// Mitsubishi GX Works2 project: atuo   PLC: FX3U/FX3UC

PROGRAM MAIN
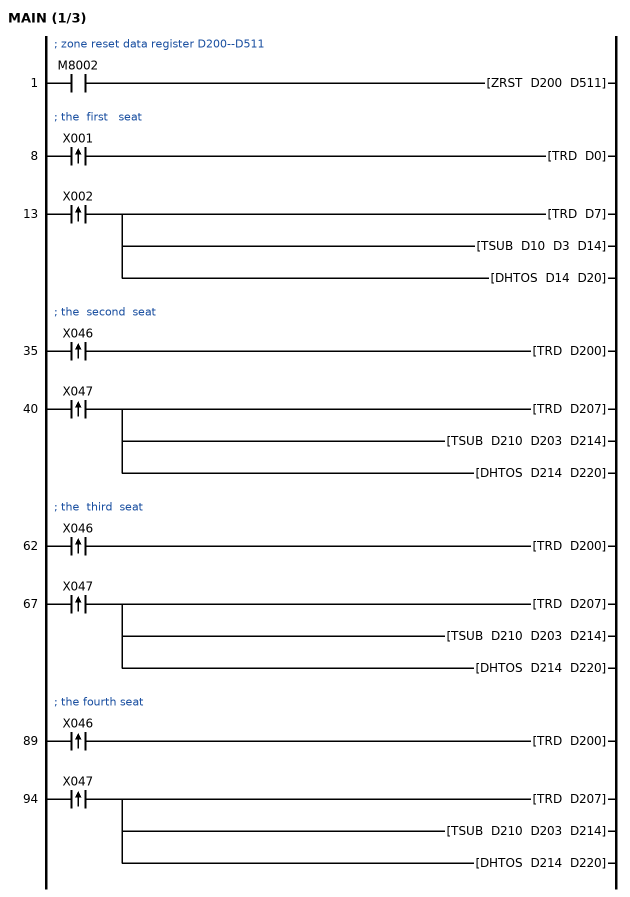
; zone reset data register D200--D511
1     LD      M8002
      ZRST    D200 D511
; the  first   seat
8     LDP     X001
      TRD     D0
13    LDP     X002
      TRD     D7
      TSUB    D10 D3 D14
      DHTOS   D14 D20
; the  second  seat
35    LDP     X046
      TRD     D200
40    LDP     X047
      TRD     D207
      TSUB    D210 D203 D214
      DHTOS   D214 D220
; the  third  seat
62    LDP     X046
      TRD     D200
67    LDP     X047
      TRD     D207
      TSUB    D210 D203 D214
      DHTOS   D214 D220
; the fourth seat
89    LDP     X046
      TRD     D200
94    LDP     X047
      TRD     D207
      TSUB    D210 D203 D214
      DHTOS   D214 D220
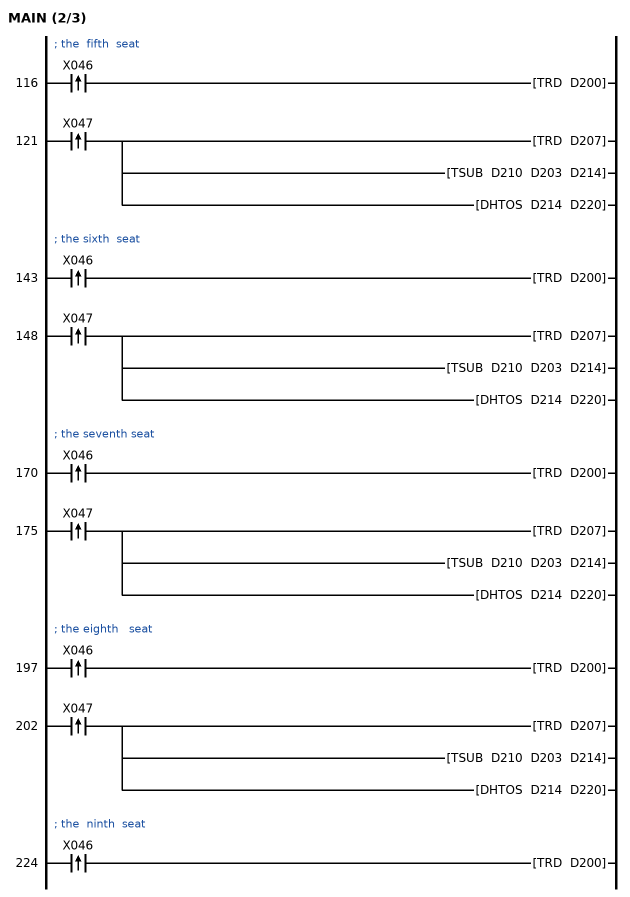
; the  fifth  seat
116   LDP     X046
      TRD     D200
121   LDP     X047
      TRD     D207
      TSUB    D210 D203 D214
      DHTOS   D214 D220
; the sixth  seat
143   LDP     X046
      TRD     D200
148   LDP     X047
      TRD     D207
      TSUB    D210 D203 D214
      DHTOS   D214 D220
; the seventh seat
170   LDP     X046
      TRD     D200
175   LDP     X047
      TRD     D207
      TSUB    D210 D203 D214
      DHTOS   D214 D220
; the eighth   seat
197   LDP     X046
      TRD     D200
202   LDP     X047
      TRD     D207
      TSUB    D210 D203 D214
      DHTOS   D214 D220
; the  ninth  seat
224   LDP     X046
      TRD     D200
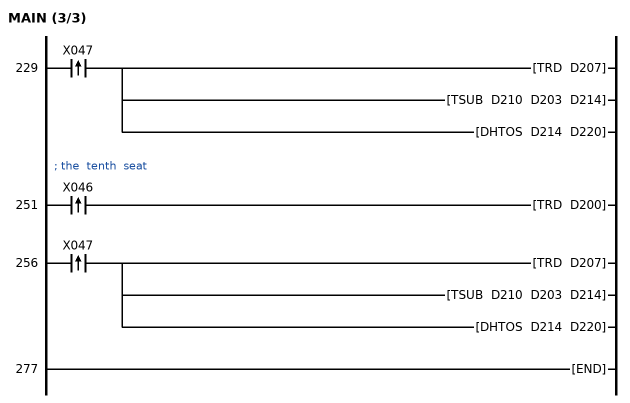
229   LDP     X047
      TRD     D207
      TSUB    D210 D203 D214
      DHTOS   D214 D220
; the  tenth  seat
251   LDP     X046
      TRD     D200
256   LDP     X047
      TRD     D207
      TSUB    D210 D203 D214
      DHTOS   D214 D220
277   END
END_PROGRAM
